// TIA Portal V20 export
TYPE "LBP_typeModularMcpAxisOutput"
TITLE = Modular MCP image / Image MCP modulaire
// Output image of axis keypad for modular MCP / Image des sorties du champ de touches d'axe pour MCP modulaires
   STRUCT
      minus : Bool;   // output image n+0 bit 0 / Image des sorties n+0 bit 0
      rapidTraverse : Bool;   // output image n+0 bit 1 / Image des sorties n+0 bit 1
      plus : Bool;   // output image n+0 bit 2 / Image des sorties n+0 bit 2
      led3 : Bool;   // output image n+0 bit 3 / Image des sorties n+0 bit 3
      tcs : Bool;   // output image n+0 bit 4 / Image des sorties n+0 bit 4
      mcsWcs : Bool;   // output image n+0 bit 5 / Image des sorties n+0 bit 5
      led6 : Bool;   // output image n+0 bit 6 / Image des sorties n+0 bit 6
      led7 : Bool;   // output image n+0 bit 7 / Image des sorties n+0 bit 7
      led8 : Bool;   // output image n+1 bit 0 / Image des sorties n+1 bit 0
      axis4 : Bool;   // output image n+1 bit 1 / Image des sorties n+1 bit 1
      axis5 : Bool;   // output image n+1 bit 2 / Image des sorties n+1 bit 2
      axis6 : Bool;   // output image n+1 bit 3 / Image des sorties n+1 bit 3
      axisX : Bool;   // output image n+1 bit 4 / Image des sorties n+1 bit 4
      axisY : Bool;   // output image n+1 bit 5 / Image des sorties n+1 bit 5
      axisZ : Bool;   // output image n+1 bit 6 / Image des sorties n+1 bit 6
      reserved17 : Bool;
      feedrateStop : Bool;   // output image n+2 bit 0 / Image des sorties n+2 bit 0
      feedrateStart : Bool;   // output image n+2 bit 1 / Image des sorties n+2 bit 1
      led18 : Bool;   // output image n+2 bit 2 / Image des sorties n+2 bit 2
      reserved23 : Bool;
      reserved24 : Bool;
      reserved25 : Bool;
      reserved26 : Bool;
      reserved27 : Bool;
      spindleStop : Bool;   // output image n+3 bit 0 / Image des sorties n+3 bit 0
      spindleStart : Bool;   // output image n+3 bit 1 / Image des sorties n+3 bit 1
      led26 : Bool;   // output image n+3 bit 2 / Image des sorties n+3 bit 2
      reserved33 : Bool;
      reserved34 : Bool;
      reserved35 : Bool;
      reserved36 : Bool;
      reserved37 : Bool;
   END_STRUCT;
END_TYPE
